// TIA Portal project "w1_B3_2DoiChoi" (V14)

(* hardware
DEVICE "S7-1200 station_1"  S7-1200 Station
   slot 0: "Rack_0"  S7-1200 Rack  Rack  V1.0
   slot 1: "PLC_1"  CPU 1214C DC/DC/DC  6ES7 214-1AG40-0XB0  V4.2
*)

// ===== PLC "PLC_1"  CPU 1214C DC/DC/DC =====

VAR_GLOBAL   // PLC tag table "Default tag table"
   "Start" AT %I0.0 : Bool;
   "B1" AT %I0.1 : Bool;
   "B2" AT %I0.2 : Bool;
   "Sig1" AT %M0.0 : Bool;
   "Sig2" AT %M0.1 : Bool;
   "D1" AT %Q0.0 : Bool;
   "D2" AT %Q0.1 : Bool;
   "Bao1" AT %Q0.2 : Bool;
   "Bao2" AT %Q0.3 : Bool;
   "rs1" AT %M0.2 : Bool;
   "rs2" AT %M0.3 : Bool;
   "ngat1" AT %M0.4 : Bool;
   "ngat2" AT %M0.5 : Bool;
   "reset" AT %I0.3 : Bool;
END_VAR

// folder: System blocks/Program resources

DATA_BLOCK "IEC_Timer_0_DB"   // DB1
{ S7_Optimized_Access := 'TRUE' }
AUTHOR : Simatic
FAMILY : IEC
NAME : IEC_TMR
VERSION : 1.0
// stored: InstanceOfName IEC_TIMER
"IEC_TIMER"
BEGIN
END_DATA_BLOCK

DATA_BLOCK "IEC_Timer_0_DB_1"   // DB2
{ S7_Optimized_Access := 'TRUE' }
AUTHOR : Simatic
FAMILY : IEC
NAME : IEC_TMR
VERSION : 1.0
// stored: InstanceOfName IEC_TIMER
"IEC_TIMER"
BEGIN
END_DATA_BLOCK

DATA_BLOCK "IEC_Timer_0_DB_2"   // DB3
{ S7_Optimized_Access := 'TRUE' }
AUTHOR : Simatic
FAMILY : IEC
NAME : IEC_TMR
VERSION : 1.0
// stored: InstanceOfName IEC_TIMER
"IEC_TIMER"
BEGIN
END_DATA_BLOCK

DATA_BLOCK "IEC_Timer_0_DB_3"   // DB4
{ S7_Optimized_Access := 'TRUE' }
AUTHOR : Simatic
FAMILY : IEC
NAME : IEC_TMR
VERSION : 1.0
// stored: InstanceOfName IEC_TIMER
"IEC_TIMER"
BEGIN
END_DATA_BLOCK

DATA_BLOCK "IEC_Timer_0_DB_4"   // DB5
{ S7_Optimized_Access := 'TRUE' }
AUTHOR : Simatic
FAMILY : IEC
NAME : IEC_TMR
VERSION : 1.0
// stored: InstanceOfName IEC_TIMER
"IEC_TIMER"
BEGIN
END_DATA_BLOCK

// folder: (top level)

ORGANIZATION_BLOCK "Main"   // OB1, LAD, ProgramCycle
TITLE = "Main Program Sweep (Cycle)"
{ S7_Optimized_Access := 'TRUE' }
VERSION : 0.1
   VAR_INPUT
      Initial_Call : Bool;   // Initial call of this OB
      Remanence : Bool;   // =True, if remanent data are available
   END_VAR
   VAR_TEMP   // added for the SCL form of the ladder/FBD networks
      _w1 : Bool;
      _w2 : Bool;
   END_VAR
BEGIN

REGION Network 1
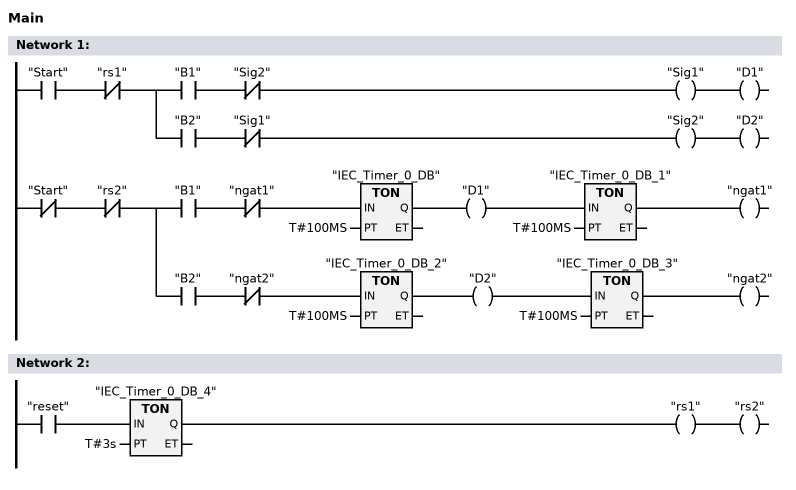
   #_w1 := "Start" AND NOT "rs1";
   "Sig1" := #_w1 AND "B1" AND NOT "Sig2";
   "D1" := "Sig1";
   "Sig2" := #_w1 AND "B2" AND NOT "Sig1";
   "D2" := "Sig2";
   #_w2 := NOT "Start" AND NOT "rs2";
   "IEC_Timer_0_DB".TON(IN := #_w2 AND "B1" AND NOT "ngat1", PT := T#100MS);
   "D1" := "IEC_Timer_0_DB".Q;
   "IEC_Timer_0_DB_1".TON(IN := "IEC_Timer_0_DB".Q, PT := T#100MS);
   "ngat1" := "IEC_Timer_0_DB_1".Q;
   "IEC_Timer_0_DB_2".TON(IN := #_w2 AND "B2" AND NOT "ngat2", PT := T#100MS);
   "D2" := "IEC_Timer_0_DB_2".Q;
   "IEC_Timer_0_DB_3".TON(IN := "IEC_Timer_0_DB_2".Q, PT := T#100MS);
   "ngat2" := "IEC_Timer_0_DB_3".Q;
END_REGION

REGION Network 2
   "IEC_Timer_0_DB_4".TON(IN := "reset", PT := T#3s);
   "rs1" := "IEC_Timer_0_DB_4".Q;
   "rs2" := "IEC_Timer_0_DB_4".Q;
END_REGION
END_ORGANIZATION_BLOCK